(* PLC project Tc2_Utilities.FB_TzSpecificLocalTimeToFileTime64 Demo, tc3-libraries-kb TwinCAT 3.1 *)
(* stored: creationDateTime 2026-05-10T20:00:00, modificationDateTime 2026-05-10T20:00:00 *)

PROGRAM P_Demo_FB_TzSpecificLocalTimeToFileTime64
  VAR
    fbFB_TzSpecificLocalTimeToFileTime64 : FB_TzSpecificLocalTimeToFileTime64;  (* Tc2_Utilities.FB_TzSpecificLocalTimeToFileTime64 实例 *)
    arg_in : T_FILETIME64;  (* VAR_INPUT in *)
    arg_tzInfo : ST_TimeZoneInformation;  (* VAR_INPUT tzInfo *)
    out_out : T_FILETIME64;  (* VAR_OUTPUT out *)
    out_eTzID : E_TimeZoneID;  (* VAR_OUTPUT eTzID *)
    out_bB : BOOL;  (* VAR_OUTPUT bB *)
  END_VAR

            // ============================================================
// Tc2_Utilities.FB_TzSpecificLocalTimeToFileTime64 演示程序（FB 实例）
// ============================================================
// 验证步骤：
//   1. 引用 Tc2_Utilities（及依赖类型所在库 Tc2_System 等）
//   2. 编译 + 登录
//   3. 按 doc.md 给 arg_* 赋值
//   4. 在线监视 out_* / io_* 输出
// ============================================================

fbFB_TzSpecificLocalTimeToFileTime64(
    in := arg_in,
    tzInfo := arg_tzInfo,
    out => out_out,
    eTzID => out_eTzID,
    bB => out_bB
);

          
END_PROGRAM
